{attribute 'qualified_only'}
VAR_GLOBAL
	nEventsInEventLogger : INT; // Number of events on event logger buffer
END_VAR

(* stored: Version 1.1.0.1, ProductVersion 3.1.4024.10
   GVL UtilityVariables: Id {c280ec43-4532-44eb-ac84-f3385987dca7} *)
